# EPICS autosave request: softGlueApp/Db/BUFFER_settings.req
$(P)$(H)BUFFER-$(N)_desc
$(P)$(H)BUFFER-$(N)_IN_Signal
$(P)$(H)BUFFER-$(N)_OUT_Signal
